Yaskawa INFORM job: u_angleTRJ0.JBI

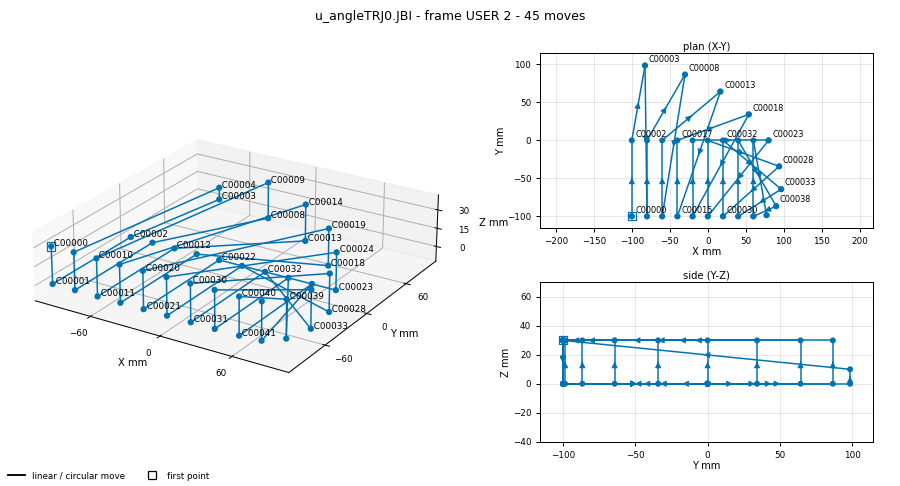
[picture p0: tool path of u_angleTRJ0.JBI in frame USER 2, 45 of 45 moves have a stored position in this frame; points joined in program order, loops and branches not executed]
/JOB
//NAME u_angleTRJ0
///FOLDERNAME DEMO
//POS
///NPOS 45,0,0,0,0,0
///USER 2
///TOOL 7
///POSTYPE USER
///RECTAN
///RCONF 1,0,0,0,0,0,0,0,0,0,0,0,0,0,0,0,0,0,0,0,0,0,0,0
C00000=-100.000,-100.000,30.000,-180.0000,-0.0000,0.0000
C00001=-100.000,-100.000,0.000,-180.0000,-0.0000,0.0000
C00002=-100.000,0.000,0.000,-180.0000,-0.0000,0.0000
C00003=-82.600,98.500,0.000,-180.0000,-0.0000,0.0000
C00004=-82.600,98.500,10.000,-180.0000,-0.0000,0.0000
C00005=-80.000,-100.000,30.000,-180.0000,-0.0000,0.0000
C00006=-80.000,-100.000,0.000,-180.0000,-0.0000,0.0000
C00007=-80.000,0.000,0.000,-180.0000,-0.0000,0.0000
C00008=-30.000,86.600,0.000,-180.0000,-0.0000,0.0000
C00009=-30.000,86.600,30.000,-180.0000,-0.0000,0.0000
C00010=-60.000,-100.000,30.000,-180.0000,-0.0000,0.0000
C00011=-60.000,-100.000,0.000,-180.0000,-0.0000,0.0000
C00012=-60.000,0.000,0.000,-180.0000,-0.0000,0.0000
C00013=16.600,64.280,0.000,-180.0000,-0.0000,0.0000
C00014=16.600,64.280,30.000,-180.0000,-0.0000,0.0000
C00015=-40.000,-100.000,30.000,-180.0000,-0.0000,0.0000
C00016=-40.000,-100.000,0.000,-180.0000,-0.0000,0.0000
C00017=-40.000,0.000,0.000,-180.0000,-0.0000,0.0000
C00018=53.970,34.200,0.000,-180.0000,-0.0000,0.0000
C00019=53.970,34.200,30.000,-180.0000,-0.0000,0.0000
C00020=-20.000,-100.000,30.000,-180.0000,-0.0000,0.0000
C00021=-20.000,-100.000,0.000,-180.0000,-0.0000,0.0000
C00022=-20.000,0.000,0.000,-180.0000,-0.0000,0.0000
C00023=80.000,0.000,0.000,-180.0000,-0.0000,0.0000
C00024=80.000,0.000,30.000,-180.0000,-0.0000,0.0000
C00025=-0.000,-100.000,30.000,-180.0000,-0.0000,0.0000
C00026=-0.000,-100.000,0.000,-180.0000,-0.0000,0.0000
C00027=-0.000,0.000,0.000,-180.0000,-0.0000,0.0000
C00028=93.970,-34.200,0.000,-180.0000,-0.0000,0.0000
C00029=93.970,-34.200,30.000,-180.0000,-0.0000,0.0000
C00030=20.000,-100.000,30.000,-180.0000,-0.0000,0.0000
C00031=20.000,-100.000,0.000,-180.0000,-0.0000,0.0000
C00032=20.000,0.000,0.000,-180.0000,-0.0000,0.0000
C00033=96.600,-64.280,0.000,-180.0000,-0.0000,0.0000
C00034=96.600,-64.280,30.000,-180.0000,-0.0000,0.0000
C00035=40.000,-100.000,30.000,-180.0000,-0.0000,0.0000
C00036=40.000,-100.000,0.000,-180.0000,-0.0000,0.0000
C00037=40.000,0.000,0.000,-180.0000,-0.0000,0.0000
C00038=90.000,-86.600,0.000,-180.0000,-0.0000,0.0000
C00039=90.000,-86.600,30.000,-180.0000,-0.0000,0.0000
C00040=60.000,-100.000,30.000,-180.0000,-0.0000,0.0000
C00041=60.000,-100.000,0.000,-180.0000,-0.0000,0.0000
C00042=60.000,0.000,0.000,-180.0000,-0.0000,0.0000
C00043=77.300,-98.480,0.000,-180.0000,-0.0000,0.0000
C00044=77.300,-98.480,30.000,-180.0000,-0.0000,0.0000
//INST
///DATE 2021/09/22 13:45
///COMM
///ATTR SC,RW,RJ
////FRAME USER 2
///GROUP1 RB1
NOP
SPEED V=20.0
' 170
MOVL C00000
MOVL C00001
ARCON
MOVL C00002
MOVL C00003
ARCOF
MOVL C00004
' 150
MOVL C00005
MOVL C00006
ARCON
MOVL C00007
MOVL C00008
ARCOF
MOVL C00009
' 130
MOVL C00010
MOVL C00011
ARCON
MOVL C00012
MOVL C00013
ARCOF
MOVL C00014
' 110
MOVL C00015
MOVL C00016
ARCON
MOVL C00017
MOVL C00018
ARCOF
MOVL C00019
' 90
MOVL C00020
MOVL C00021
ARCON
MOVL C00022
MOVL C00023
ARCOF
MOVL C00024
' 70
MOVL C00025
MOVL C00026
ARCON
MOVL C00027
MOVL C00028
ARCOF
MOVL C00029
' 50
MOVL C00030
MOVL C00031
ARCON
MOVL C00032
MOVL C00033
ARCOF
MOVL C00034
' 30
MOVL C00035
MOVL C00036
ARCON
MOVL C00037
MOVL C00038
ARCOF
MOVL C00039
' 10
MOVL C00040
MOVL C00041
ARCON
MOVL C00042
MOVL C00043
ARCOF
MOVL C00044
END
